Universal Robots PolyScope program: switch_operator_input.urp

Program switch_operator_input (createdIn=3.2.18515 lastSavedIn=3.2.18515 directory=/home/ur/ursim-3.2/programs installation=default robotSerialNumber=2014359999)
Calibrated DH parameters: a=[0, -0.425, -0.39225, 0, 0, 0]; d=[0.089159, 0, 0, 0.10915, 0.09465, 0.0823]; alpha=[1.570796, 0, 0, 1.570796, -1.570796, 0]; deltaTheta=[0, 0, 0, 0, 0, 0]
Robot Program (runOnlyOnce=false motionType=MoveJ speed=1.047198 acceleration=1.396263 recalculateMotions=false)
  var_1 :=  (valueSource=Operator message=Enter a number between 1 to 4 valueType=Integer)
  Switch expression=var_1
    Case (caseValue=1)
      Popup Message (haltProgram=false message=case1)
    Case (caseValue=2)
      Popup Message (haltProgram=false message=case2)
    Case (caseValue=3)
      Popup Message (haltProgram=false message=case3)
    Case (caseValue=4)
      Popup Message (haltProgram=false message=case4)
    Case (caseValue=2147483647)
      Popup Message (haltProgram=false message=You have entered a number outside 1 to 4)
